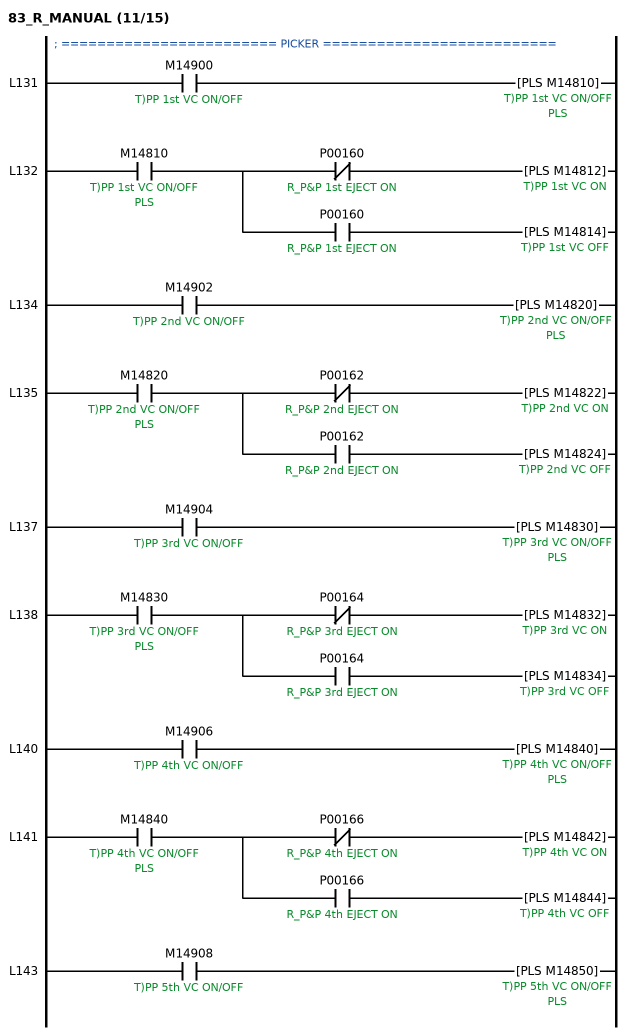
[picture p336: 83_R_MANUAL rungs L131-L143]
// ======================== PICKER ==========================
; L131
LOAD      M14900	// T)PP 1st VC ON/OFF
OUTP      M14810	// T)PP 1st VC ON/OFF PLS
; L132
LOAD      M14810	// T)PP 1st VC ON/OFF PLS
MPUSH
AND NOT   P00160	// R_P&P 1st EJECT ON
OUTP      M14812	// T)PP 1st VC ON
MPOP
AND       P00160	// R_P&P 1st EJECT ON
OUTP      M14814	// T)PP 1st VC OFF
; L134
LOAD      M14902	// T)PP 2nd VC ON/OFF
OUTP      M14820	// T)PP 2nd VC ON/OFF PLS
; L135
LOAD      M14820	// T)PP 2nd VC ON/OFF PLS
MPUSH
AND NOT   P00162	// R_P&P 2nd EJECT ON
OUTP      M14822	// T)PP 2nd VC ON
MPOP
AND       P00162	// R_P&P 2nd EJECT ON
OUTP      M14824	// T)PP 2nd VC OFF
; L137
LOAD      M14904	// T)PP 3rd VC ON/OFF
OUTP      M14830	// T)PP 3rd VC ON/OFF PLS
; L138
LOAD      M14830	// T)PP 3rd VC ON/OFF PLS
MPUSH
AND NOT   P00164	// R_P&P 3rd EJECT ON
OUTP      M14832	// T)PP 3rd VC ON
MPOP
AND       P00164	// R_P&P 3rd EJECT ON
OUTP      M14834	// T)PP 3rd VC OFF
; L140
LOAD      M14906	// T)PP 4th VC ON/OFF
OUTP      M14840	// T)PP 4th VC ON/OFF PLS
; L141
LOAD      M14840	// T)PP 4th VC ON/OFF PLS
MPUSH
AND NOT   P00166	// R_P&P 4th EJECT ON
OUTP      M14842	// T)PP 4th VC ON
MPOP
AND       P00166	// R_P&P 4th EJECT ON
OUTP      M14844	// T)PP 4th VC OFF
; L143
LOAD      M14908	// T)PP 5th VC ON/OFF
OUTP      M14850	// T)PP 5th VC ON/OFF PLS

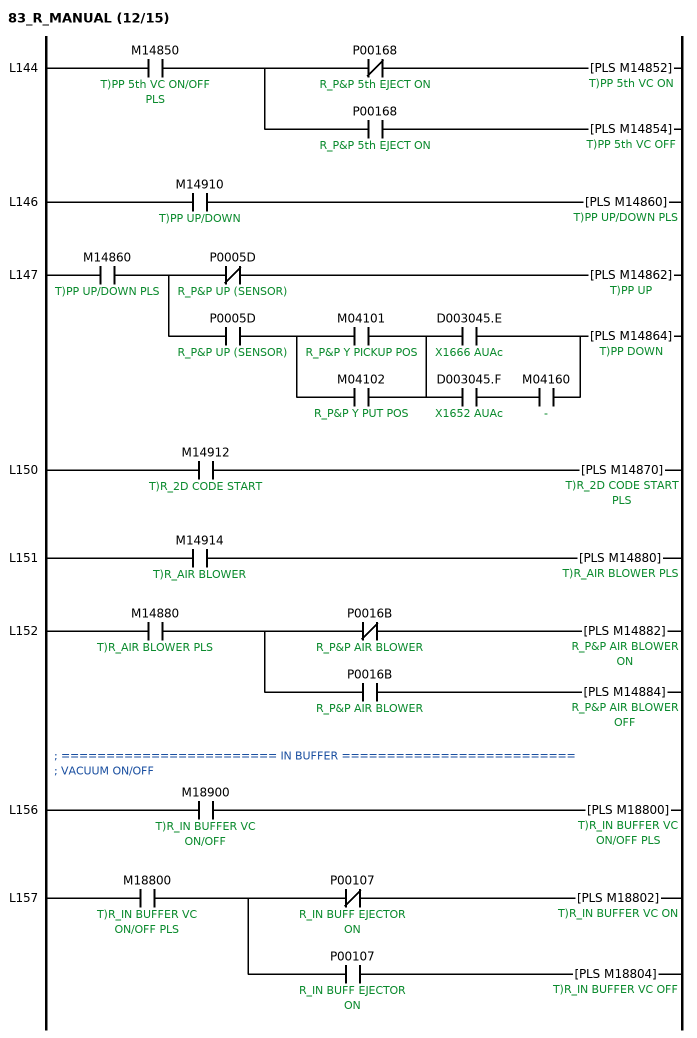
; L144
LOAD      M14850	// T)PP 5th VC ON/OFF PLS
MPUSH
AND NOT   P00168	// R_P&P 5th EJECT ON
OUTP      M14852	// T)PP 5th VC ON
MPOP
AND       P00168	// R_P&P 5th EJECT ON
OUTP      M14854	// T)PP 5th VC OFF
; L146
LOAD      M14910	// T)PP UP/DOWN
OUTP      M14860	// T)PP UP/DOWN PLS
; L147
LOAD      M14860	// T)PP UP/DOWN PLS
MPUSH
AND NOT   P0005D	// R_P&P UP (SENSOR)
OUTP      M14862	// T)PP UP
MPOP
AND       P0005D	// R_P&P UP (SENSOR)
LOAD      M04101	// R_P&P Y PICKUP POS
OR        M04102	// R_P&P Y PUT POS
AND LOAD
LOAD      D003045.E	// X1666 AUAc
LOAD      D003045.F	// X1652 AUAc
AND       M04160	// -
OR LOAD
AND LOAD
OUTP      M14864	// T)PP DOWN
; L150
LOAD      M14912	// T)R_2D CODE START
OUTP      M14870	// T)R_2D CODE START PLS
; L151
LOAD      M14914	// T)R_AIR BLOWER
OUTP      M14880	// T)R_AIR BLOWER PLS
; L152
LOAD      M14880	// T)R_AIR BLOWER PLS
MPUSH
AND NOT   P0016B	// R_P&P AIR BLOWER
OUTP      M14882	// R_P&P AIR BLOWER ON
MPOP
AND       P0016B	// R_P&P AIR BLOWER
OUTP      M14884	// R_P&P AIR BLOWER OFF
// ======================== IN BUFFER ==========================
// VACUUM ON/OFF
; L156
LOAD      M18900	// T)R_IN BUFFER VC ON/OFF
OUTP      M18800	// T)R_IN BUFFER VC ON/OFF PLS
; L157
LOAD      M18800	// T)R_IN BUFFER VC ON/OFF PLS
MPUSH
AND NOT   P00107	// R_IN BUFF EJECTOR ON
OUTP      M18802	// T)R_IN BUFFER VC ON
MPOP
AND       P00107	// R_IN BUFF EJECTOR ON
OUTP      M18804	// T)R_IN BUFFER VC OFF

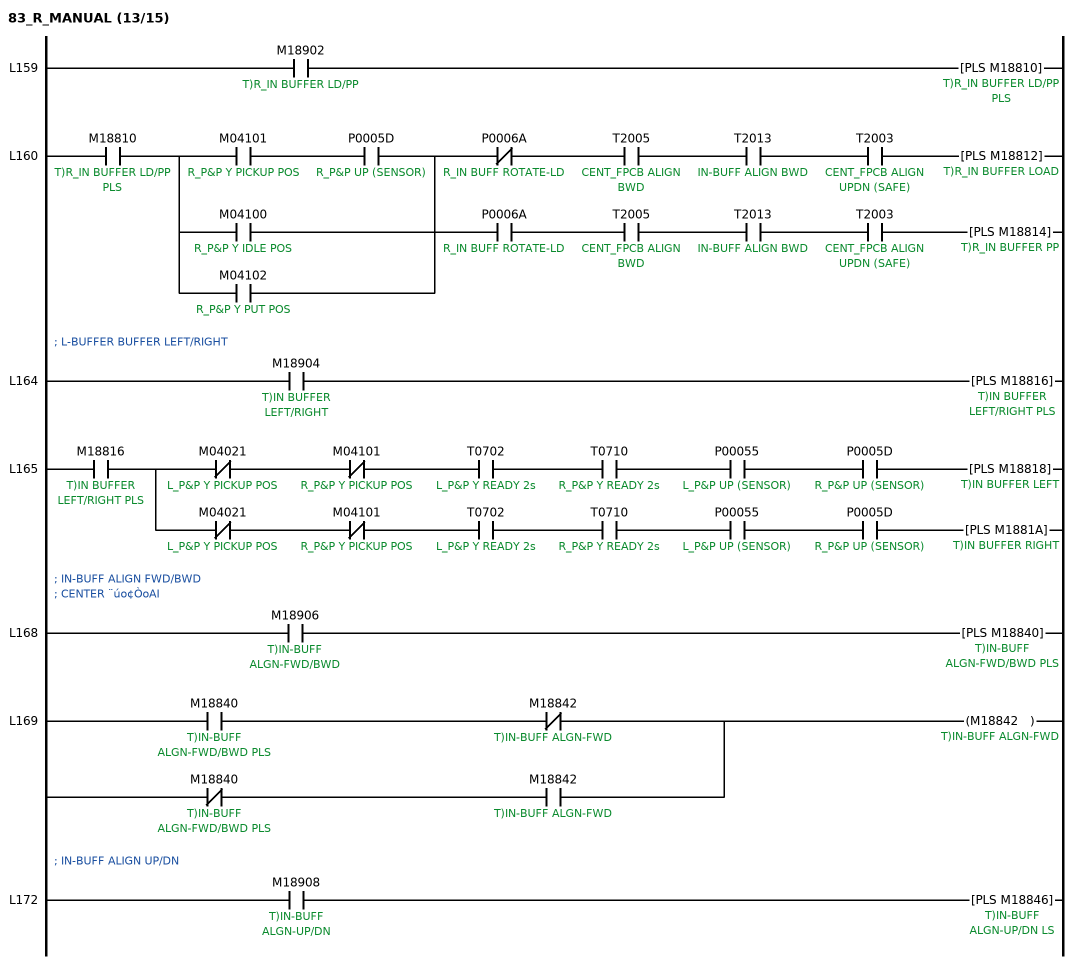
; L159
LOAD      M18902	// T)R_IN BUFFER LD/PP
OUTP      M18810	// T)R_IN BUFFER LD/PP PLS
; L160
LOAD      M18810	// T)R_IN BUFFER LD/PP PLS
LOAD      M04101	// R_P&P Y PICKUP POS
AND       P0005D	// R_P&P UP (SENSOR)
OR        M04100	// R_P&P Y IDLE POS
OR        M04102	// R_P&P Y PUT POS
AND LOAD
MPUSH
AND NOT   P0006A	// R_IN BUFF ROTATE-LD
AND       T2005	// CENT_FPCB ALIGN BWD
AND       T2013	// IN-BUFF ALIGN BWD
AND       T2003	// CENT_FPCB ALIGN UPDN (SAFE)
OUTP      M18812	// T)R_IN BUFFER LOAD
MPOP
AND       P0006A	// R_IN BUFF ROTATE-LD
AND       T2005	// CENT_FPCB ALIGN BWD
AND       T2013	// IN-BUFF ALIGN BWD
AND       T2003	// CENT_FPCB ALIGN UPDN (SAFE)
OUTP      M18814	// T)R_IN BUFFER PP
// L-BUFFER BUFFER LEFT/RIGHT
; L164
LOAD      M18904	// T)IN BUFFER LEFT/RIGHT
OUTP      M18816	// T)IN BUFFER LEFT/RIGHT PLS
; L165
LOAD      M18816	// T)IN BUFFER LEFT/RIGHT PLS
MPUSH
AND NOT   M04021	// L_P&P Y PICKUP POS
AND NOT   M04101	// R_P&P Y PICKUP POS
AND       T0702	// L_P&P Y READY 2s
AND       T0710	// R_P&P Y READY 2s
AND       P00055	// L_P&P UP (SENSOR)
AND       P0005D	// R_P&P UP (SENSOR)
OUTP      M18818	// T)IN BUFFER LEFT
MPOP
AND NOT   M04021	// L_P&P Y PICKUP POS
AND NOT   M04101	// R_P&P Y PICKUP POS
AND       T0702	// L_P&P Y READY 2s
AND       T0710	// R_P&P Y READY 2s
AND       P00055	// L_P&P UP (SENSOR)
AND       P0005D	// R_P&P UP (SENSOR)
OUTP      M1881A	// T)IN BUFFER RIGHT
// IN-BUFF ALIGN FWD/BWD
; L168
LOAD      M18906	// T)IN-BUFF ALGN-FWD/BWD
OUTP      M18840	// T)IN-BUFF ALGN-FWD/BWD PLS
// output comment: CENTER ¨úo¢ÒoAI
; L169
LOAD      M18840	// T)IN-BUFF ALGN-FWD/BWD PLS
AND NOT   M18842	// T)IN-BUFF ALGN-FWD
LOAD NOT  M18840	// T)IN-BUFF ALGN-FWD/BWD PLS
AND       M18842	// T)IN-BUFF ALGN-FWD
OR LOAD
OUT       M18842	// T)IN-BUFF ALGN-FWD
// IN-BUFF ALIGN UP/DN
; L172
LOAD      M18908	// T)IN-BUFF ALGN-UP/DN
OUTP      M18846	// T)IN-BUFF ALGN-UP/DN LS

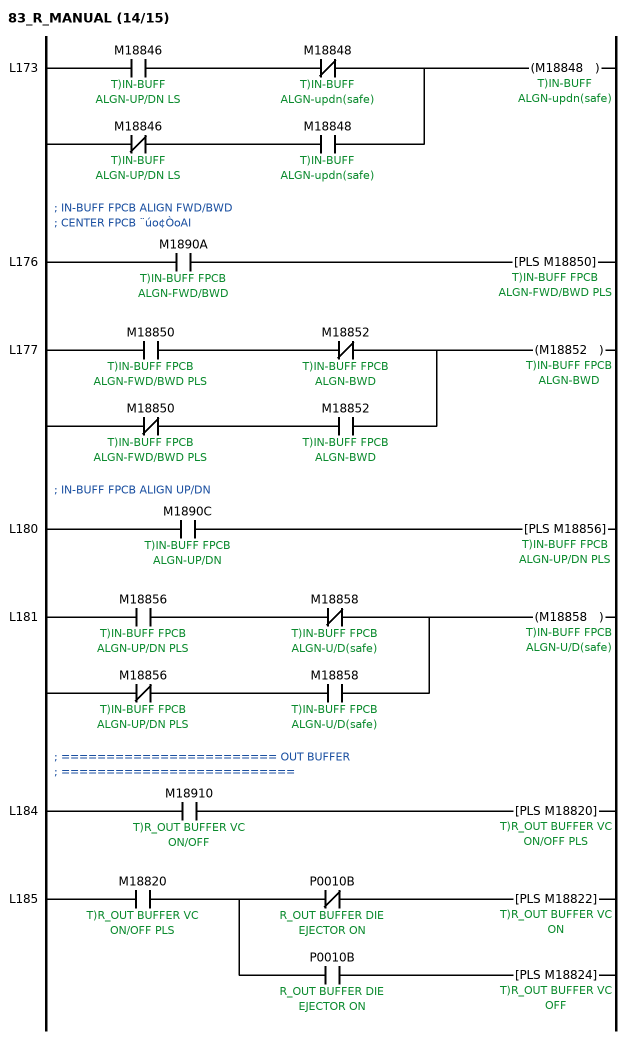
; L173
LOAD      M18846	// T)IN-BUFF ALGN-UP/DN LS
AND NOT   M18848	// T)IN-BUFF ALGN-updn(safe)
LOAD NOT  M18846	// T)IN-BUFF ALGN-UP/DN LS
AND       M18848	// T)IN-BUFF ALGN-updn(safe)
OR LOAD
OUT       M18848	// T)IN-BUFF ALGN-updn(safe)
// IN-BUFF FPCB ALIGN FWD/BWD
; L176
LOAD      M1890A	// T)IN-BUFF FPCB ALGN-FWD/BWD
OUTP      M18850	// T)IN-BUFF FPCB ALGN-FWD/BWD PLS
// output comment: CENTER FPCB ¨úo¢ÒoAI
; L177
LOAD      M18850	// T)IN-BUFF FPCB ALGN-FWD/BWD PLS
AND NOT   M18852	// T)IN-BUFF FPCB ALGN-BWD
LOAD NOT  M18850	// T)IN-BUFF FPCB ALGN-FWD/BWD PLS
AND       M18852	// T)IN-BUFF FPCB ALGN-BWD
OR LOAD
OUT       M18852	// T)IN-BUFF FPCB ALGN-BWD
// IN-BUFF FPCB ALIGN UP/DN
; L180
LOAD      M1890C	// T)IN-BUFF FPCB ALGN-UP/DN
OUTP      M18856	// T)IN-BUFF FPCB ALGN-UP/DN PLS
; L181
LOAD      M18856	// T)IN-BUFF FPCB ALGN-UP/DN PLS
AND NOT   M18858	// T)IN-BUFF FPCB ALGN-U/D(safe)
LOAD NOT  M18856	// T)IN-BUFF FPCB ALGN-UP/DN PLS
AND       M18858	// T)IN-BUFF FPCB ALGN-U/D(safe)
OR LOAD
OUT       M18858	// T)IN-BUFF FPCB ALGN-U/D(safe)
// ======================== OUT BUFFER ==========================
; L184
LOAD      M18910	// T)R_OUT BUFFER VC ON/OFF
OUTP      M18820	// T)R_OUT BUFFER VC ON/OFF PLS
; L185
LOAD      M18820	// T)R_OUT BUFFER VC ON/OFF PLS
MPUSH
AND NOT   P0010B	// R_OUT BUFFER DIE EJECTOR ON
OUTP      M18822	// T)R_OUT BUFFER VC ON
MPOP
AND       P0010B	// R_OUT BUFFER DIE EJECTOR ON
OUTP      M18824	// T)R_OUT BUFFER VC OFF

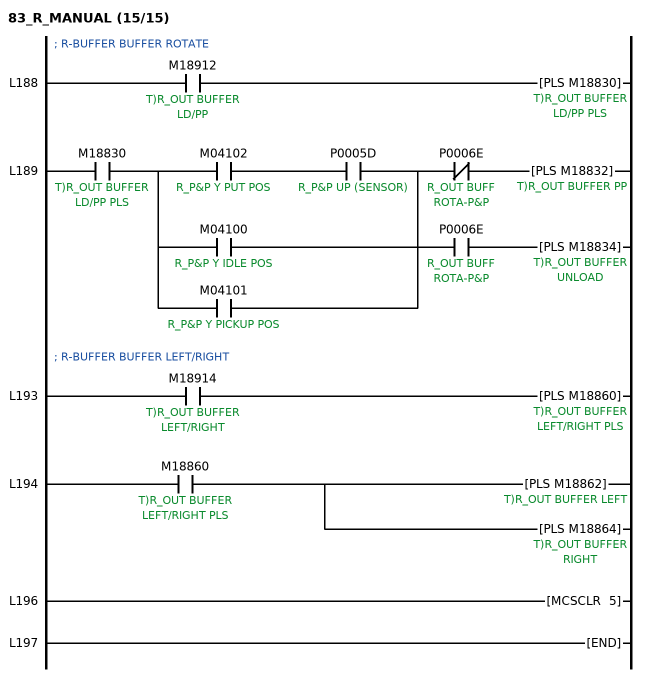
// R-BUFFER BUFFER ROTATE
; L188
LOAD      M18912	// T)R_OUT BUFFER LD/PP
OUTP      M18830	// T)R_OUT BUFFER LD/PP PLS
; L189
LOAD      M18830	// T)R_OUT BUFFER LD/PP PLS
LOAD      M04102	// R_P&P Y PUT POS
AND       P0005D	// R_P&P UP (SENSOR)
OR        M04100	// R_P&P Y IDLE POS
OR        M04101	// R_P&P Y PICKUP POS
AND LOAD
MPUSH
AND NOT   P0006E	// R_OUT BUFF ROTA-P&P
OUTP      M18832	// T)R_OUT BUFFER PP
MPOP
AND       P0006E	// R_OUT BUFF ROTA-P&P
OUTP      M18834	// T)R_OUT BUFFER UNLOAD
// R-BUFFER BUFFER LEFT/RIGHT
; L193
LOAD      M18914	// T)R_OUT BUFFER LEFT/RIGHT
OUTP      M18860	// T)R_OUT BUFFER LEFT/RIGHT PLS
; L194
LOAD      M18860	// T)R_OUT BUFFER LEFT/RIGHT PLS
OUTP      M18862	// T)R_OUT BUFFER LEFT
OUTP      M18864	// T)R_OUT BUFFER RIGHT
; L196
MCSCLR    5
; L197
END

PROGRAM 84_RUN_TIME (task: ¨ö¨¬A¥ì CA¡¤I¡¾¡¿¡¤¡Í)

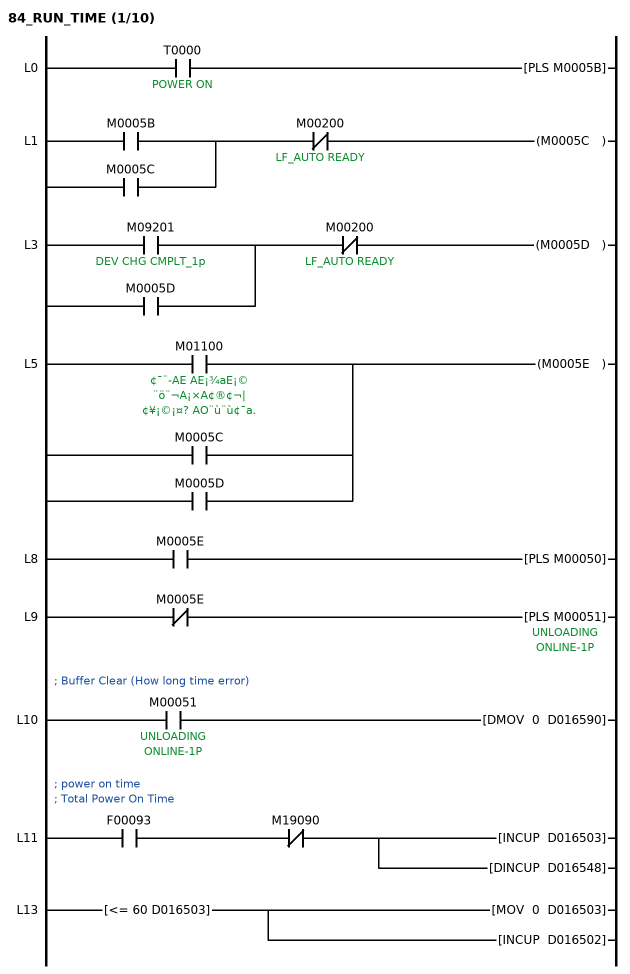
; L0
LOAD      T0000	// POWER ON
OUTP      M0005B
; L1
LOAD      M0005B
OR        M0005C
AND NOT   M00200	// LF_AUTO READY
OUT       M0005C
; L3
LOAD      M09201	// DEV CHG CMPLT_1p
OR        M0005D
AND NOT   M00200	// LF_AUTO READY
OUT       M0005D
; L5
LOAD      M01100	// ¢¯¨­AE AE¡¾aE¡© ¨ö¨¬A¡×A¢®¢¬| ¢¥¡©¡¤? AO¨ù¨ù¢¯a.
OR        M0005C
OR        M0005D
OUT       M0005E
; L8
LOAD      M0005E
OUTP      M00050
; L9
LOAD NOT  M0005E
OUTP      M00051	// UNLOADING ONLINE-1P
; L10
LOAD      M00051	// UNLOADING ONLINE-1P
DMOV      0 D016590
// output comment: Buffer Clear (How long time error)
; L11
LOAD      F00093
AND NOT   M19090
INCUP     D016503
DINCUP    D016548
// output comment: power on time
// output comment: Total Power On Time
; L13
LOAD<=    60 D016503
MOV       0 D016503
INCUP     D016502

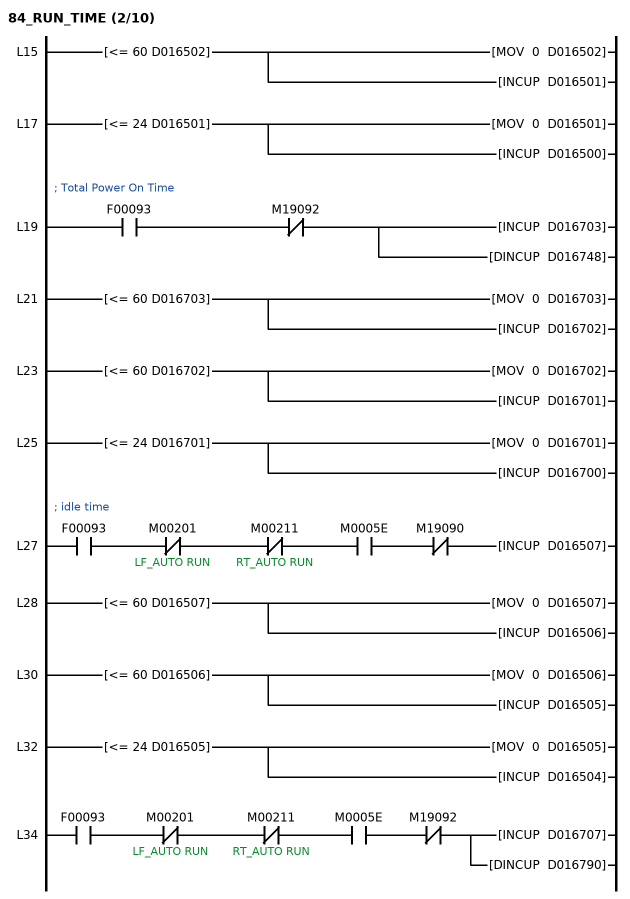
; L15
LOAD<=    60 D016502
MOV       0 D016502
INCUP     D016501
; L17
LOAD<=    24 D016501
MOV       0 D016501
INCUP     D016500
; L19
LOAD      F00093
AND NOT   M19092
INCUP     D016703
DINCUP    D016748
// output comment: Total Power On Time
; L21
LOAD<=    60 D016703
MOV       0 D016703
INCUP     D016702
; L23
LOAD<=    60 D016702
MOV       0 D016702
INCUP     D016701
; L25
LOAD<=    24 D016701
MOV       0 D016701
INCUP     D016700
; L27
LOAD      F00093
AND NOT   M00201	// LF_AUTO RUN
AND NOT   M00211	// RT_AUTO RUN
AND       M0005E
AND NOT   M19090
INCUP     D016507
// output comment: idle time
; L28
LOAD<=    60 D016507
MOV       0 D016507
INCUP     D016506
; L30
LOAD<=    60 D016506
MOV       0 D016506
INCUP     D016505
; L32
LOAD<=    24 D016505
MOV       0 D016505
INCUP     D016504
; L34
LOAD      F00093
AND NOT   M00201	// LF_AUTO RUN
AND NOT   M00211	// RT_AUTO RUN
AND       M0005E
AND NOT   M19092
INCUP     D016707
DINCUP    D016790

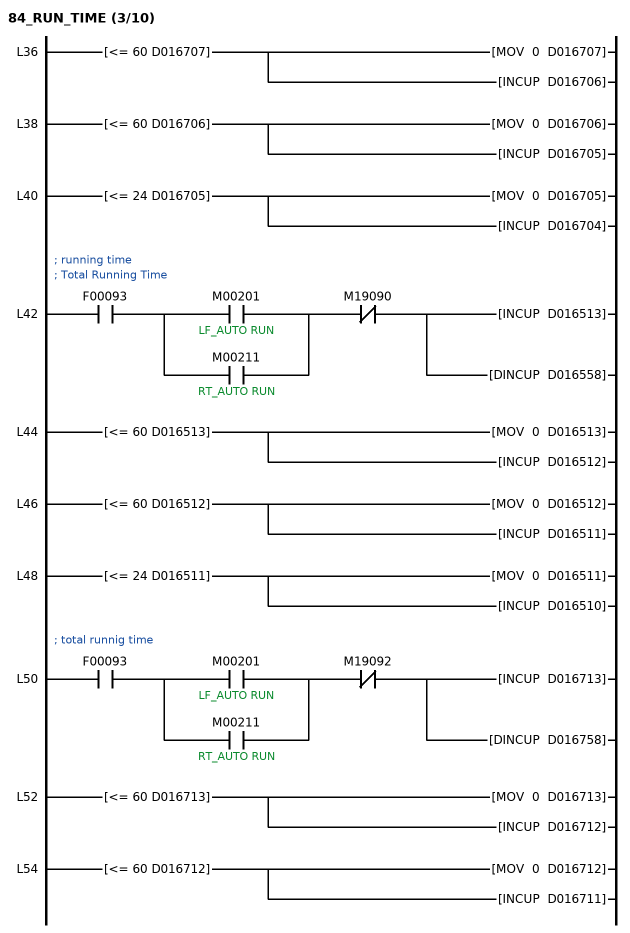
; L36
LOAD<=    60 D016707
MOV       0 D016707
INCUP     D016706
; L38
LOAD<=    60 D016706
MOV       0 D016706
INCUP     D016705
; L40
LOAD<=    24 D016705
MOV       0 D016705
INCUP     D016704
; L42
LOAD      F00093
LOAD      M00201	// LF_AUTO RUN
OR        M00211	// RT_AUTO RUN
AND LOAD
AND NOT   M19090
INCUP     D016513
DINCUP    D016558
// output comment: running time
// output comment: Total Running Time
; L44
LOAD<=    60 D016513
MOV       0 D016513
INCUP     D016512
; L46
LOAD<=    60 D016512
MOV       0 D016512
INCUP     D016511
; L48
LOAD<=    24 D016511
MOV       0 D016511
INCUP     D016510
; L50
LOAD      F00093
LOAD      M00201	// LF_AUTO RUN
OR        M00211	// RT_AUTO RUN
AND LOAD
AND NOT   M19092
INCUP     D016713
DINCUP    D016758
// output comment: total runnig time
; L52
LOAD<=    60 D016713
MOV       0 D016713
INCUP     D016712
; L54
LOAD<=    60 D016712
MOV       0 D016712
INCUP     D016711

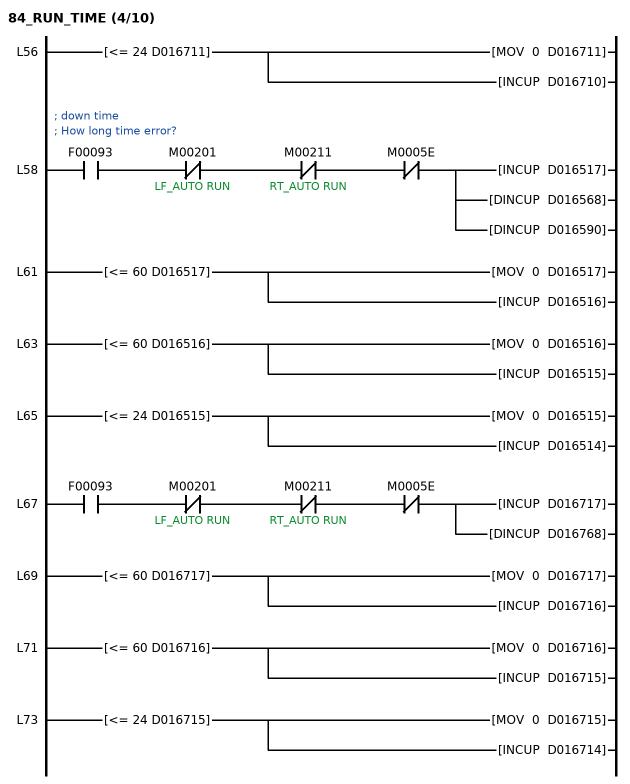
; L56
LOAD<=    24 D016711
MOV       0 D016711
INCUP     D016710
; L58
LOAD      F00093
AND NOT   M00201	// LF_AUTO RUN
AND NOT   M00211	// RT_AUTO RUN
AND NOT   M0005E
INCUP     D016517
DINCUP    D016568
DINCUP    D016590
// output comment: down time
// output comment: How long time error?
; L61
LOAD<=    60 D016517
MOV       0 D016517
INCUP     D016516
; L63
LOAD<=    60 D016516
MOV       0 D016516
INCUP     D016515
; L65
LOAD<=    24 D016515
MOV       0 D016515
INCUP     D016514
; L67
LOAD      F00093
AND NOT   M00201	// LF_AUTO RUN
AND NOT   M00211	// RT_AUTO RUN
AND NOT   M0005E
INCUP     D016717
DINCUP    D016768
; L69
LOAD<=    60 D016717
MOV       0 D016717
INCUP     D016716
; L71
LOAD<=    60 D016716
MOV       0 D016716
INCUP     D016715
; L73
LOAD<=    24 D016715
MOV       0 D016715
INCUP     D016714

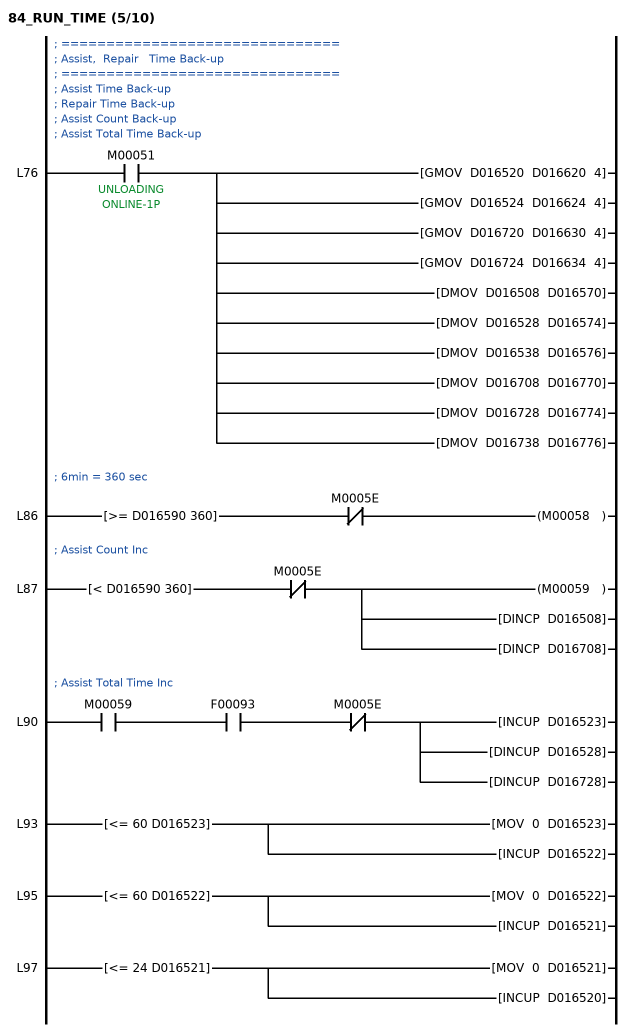
// ===============================
// Assist,  Repair   Time Back-up
// ===============================
; L76
LOAD      M00051	// UNLOADING ONLINE-1P
GMOV      D016520 D016620 4
GMOV      D016524 D016624 4
GMOV      D016720 D016630 4
GMOV      D016724 D016634 4
DMOV      D016508 D016570
DMOV      D016528 D016574
DMOV      D016538 D016576
DMOV      D016708 D016770
DMOV      D016728 D016774
DMOV      D016738 D016776
// output comment: Assist Time Back-up
// output comment: Repair Time Back-up
// output comment: Assist Count Back-up
// output comment: Assist Total Time Back-up
; L86
LOAD>=    D016590 360
AND NOT   M0005E
OUT       M00058
// output comment: 6min = 360 sec
; L87
LOAD<     D016590 360
AND NOT   M0005E
OUT       M00059
DINCP     D016508
DINCP     D016708
// output comment: Assist Count Inc
; L90
LOAD      M00059
AND       F00093
AND NOT   M0005E
INCUP     D016523
DINCUP    D016528
DINCUP    D016728
// output comment: Assist Total Time Inc
; L93
LOAD<=    60 D016523
MOV       0 D016523
INCUP     D016522
; L95
LOAD<=    60 D016522
MOV       0 D016522
INCUP     D016521
; L97
LOAD<=    24 D016521
MOV       0 D016521
INCUP     D016520

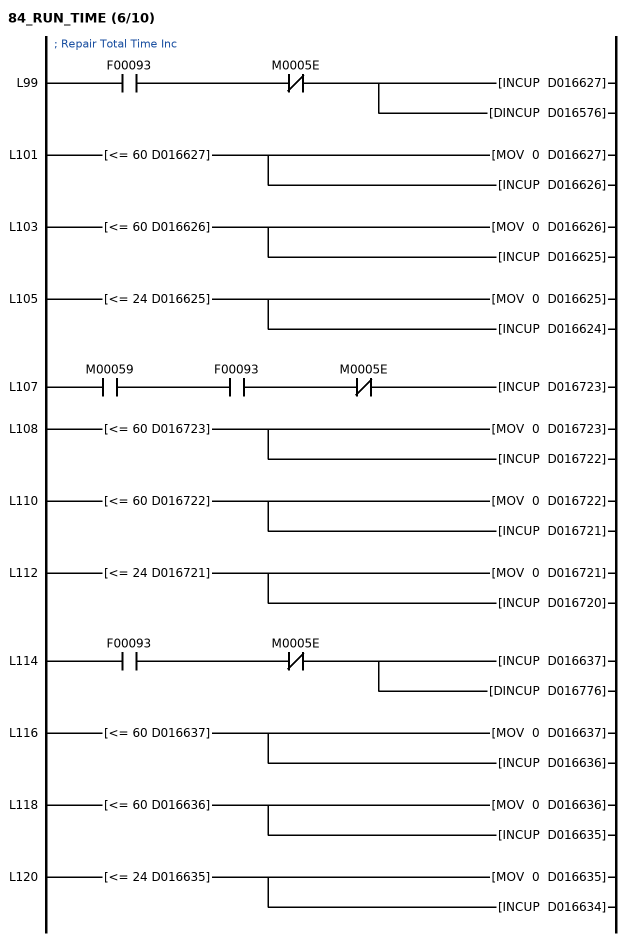
; L99
LOAD      F00093
AND NOT   M0005E
INCUP     D016627
DINCUP    D016576
// output comment: Repair Total Time Inc
; L101
LOAD<=    60 D016627
MOV       0 D016627
INCUP     D016626
; L103
LOAD<=    60 D016626
MOV       0 D016626
INCUP     D016625
; L105
LOAD<=    24 D016625
MOV       0 D016625
INCUP     D016624
; L107
LOAD      M00059
AND       F00093
AND NOT   M0005E
INCUP     D016723
; L108
LOAD<=    60 D016723
MOV       0 D016723
INCUP     D016722
; L110
LOAD<=    60 D016722
MOV       0 D016722
INCUP     D016721
; L112
LOAD<=    24 D016721
MOV       0 D016721
INCUP     D016720
; L114
LOAD      F00093
AND NOT   M0005E
INCUP     D016637
DINCUP    D016776
; L116
LOAD<=    60 D016637
MOV       0 D016637
INCUP     D016636
; L118
LOAD<=    60 D016636
MOV       0 D016636
INCUP     D016635
; L120
LOAD<=    24 D016635
MOV       0 D016635
INCUP     D016634

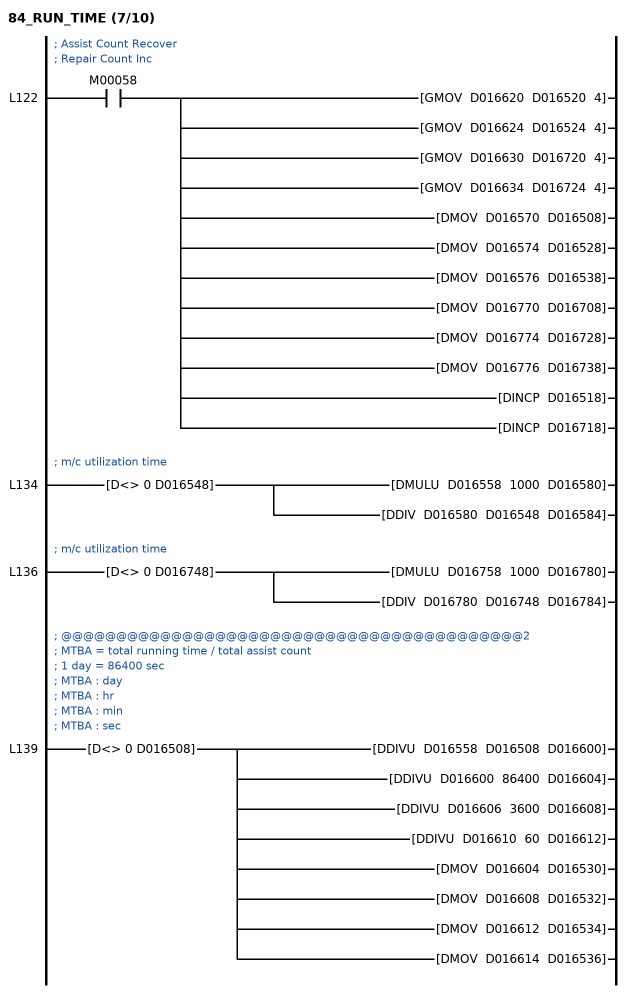
; L122
LOAD      M00058
GMOV      D016620 D016520 4
GMOV      D016624 D016524 4
GMOV      D016630 D016720 4
GMOV      D016634 D016724 4
DMOV      D016570 D016508
DMOV      D016574 D016528
DMOV      D016576 D016538
DMOV      D016770 D016708
DMOV      D016774 D016728
DMOV      D016776 D016738
DINCP     D016518
DINCP     D016718
// output comment: Assist Count Recover
// output comment: Repair Count Inc
; L134
LOADD<>   0 D016548
DMULU     D016558 1000 D016580
DDIV      D016580 D016548 D016584
// output comment: m/c utilization time
; L136
LOADD<>   0 D016748
DMULU     D016758 1000 D016780
DDIV      D016780 D016748 D016784
// output comment: m/c utilization time
// @@@@@@@@@@@@@@@@@@@@@@@@@@@@@@@@@@@@@@@@@@2
; L139
LOADD<>   0 D016508
DDIVU     D016558 D016508 D016600
DDIVU     D016600 86400 D016604
DDIVU     D016606 3600 D016608
DDIVU     D016610 60 D016612
DMOV      D016604 D016530
DMOV      D016608 D016532
DMOV      D016612 D016534
DMOV      D016614 D016536
// output comment: MTBA = total running time / total assist count
// output comment: 1 day = 86400 sec
// output comment: MTBA : day
// output comment: MTBA : hr
// output comment: MTBA : min
// output comment: MTBA : sec

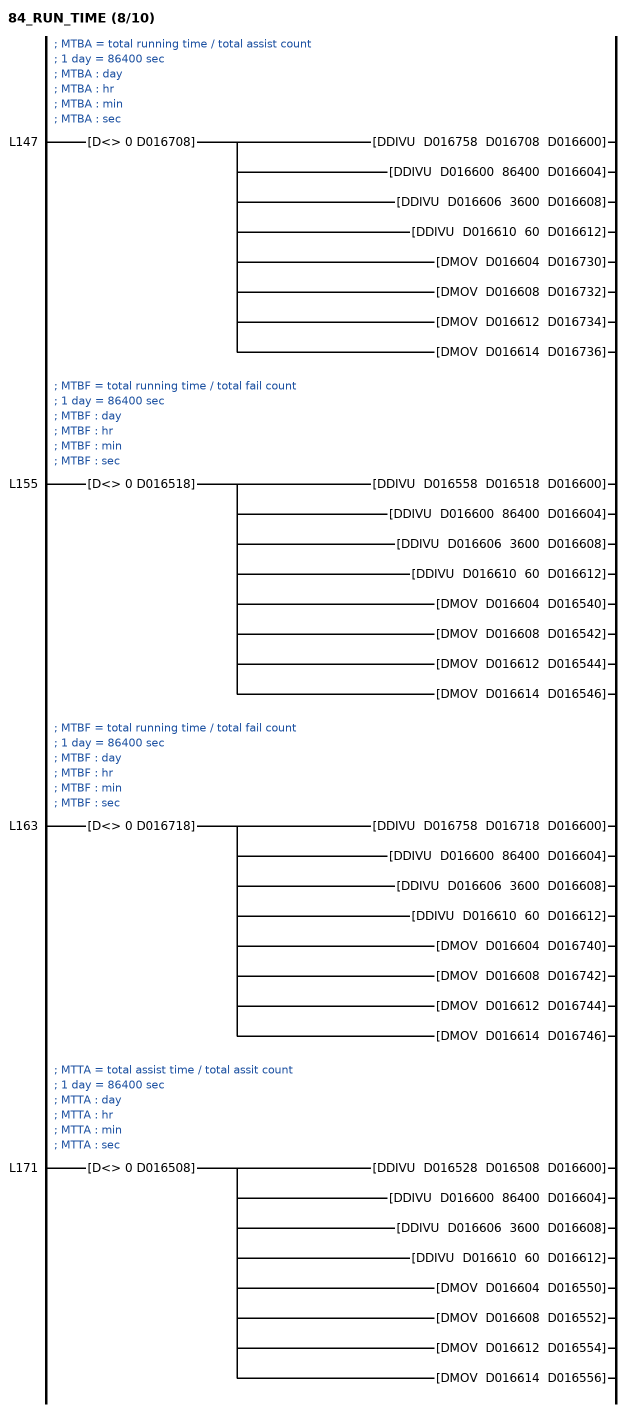
; L147
LOADD<>   0 D016708
DDIVU     D016758 D016708 D016600
DDIVU     D016600 86400 D016604
DDIVU     D016606 3600 D016608
DDIVU     D016610 60 D016612
DMOV      D016604 D016730
DMOV      D016608 D016732
DMOV      D016612 D016734
DMOV      D016614 D016736
// output comment: MTBA = total running time / total assist count
// output comment: 1 day = 86400 sec
// output comment: MTBA : day
// output comment: MTBA : hr
// output comment: MTBA : min
// output comment: MTBA : sec
; L155
LOADD<>   0 D016518
DDIVU     D016558 D016518 D016600
DDIVU     D016600 86400 D016604
DDIVU     D016606 3600 D016608
DDIVU     D016610 60 D016612
DMOV      D016604 D016540
DMOV      D016608 D016542
DMOV      D016612 D016544
DMOV      D016614 D016546
// output comment: MTBF = total running time / total fail count
// output comment: 1 day = 86400 sec
// output comment: MTBF : day
// output comment: MTBF : hr
// output comment: MTBF : min
// output comment: MTBF : sec
; L163
LOADD<>   0 D016718
DDIVU     D016758 D016718 D016600
DDIVU     D016600 86400 D016604
DDIVU     D016606 3600 D016608
DDIVU     D016610 60 D016612
DMOV      D016604 D016740
DMOV      D016608 D016742
DMOV      D016612 D016744
DMOV      D016614 D016746
// output comment: MTBF = total running time / total fail count
// output comment: 1 day = 86400 sec
// output comment: MTBF : day
// output comment: MTBF : hr
// output comment: MTBF : min
// output comment: MTBF : sec
; L171
LOADD<>   0 D016508
DDIVU     D016528 D016508 D016600
DDIVU     D016600 86400 D016604
DDIVU     D016606 3600 D016608
DDIVU     D016610 60 D016612
DMOV      D016604 D016550
DMOV      D016608 D016552
DMOV      D016612 D016554
DMOV      D016614 D016556
// output comment: MTTA = total assist time / total assit count
// output comment: 1 day = 86400 sec
// output comment: MTTA : day
// output comment: MTTA : hr
// output comment: MTTA : min
// output comment: MTTA : sec

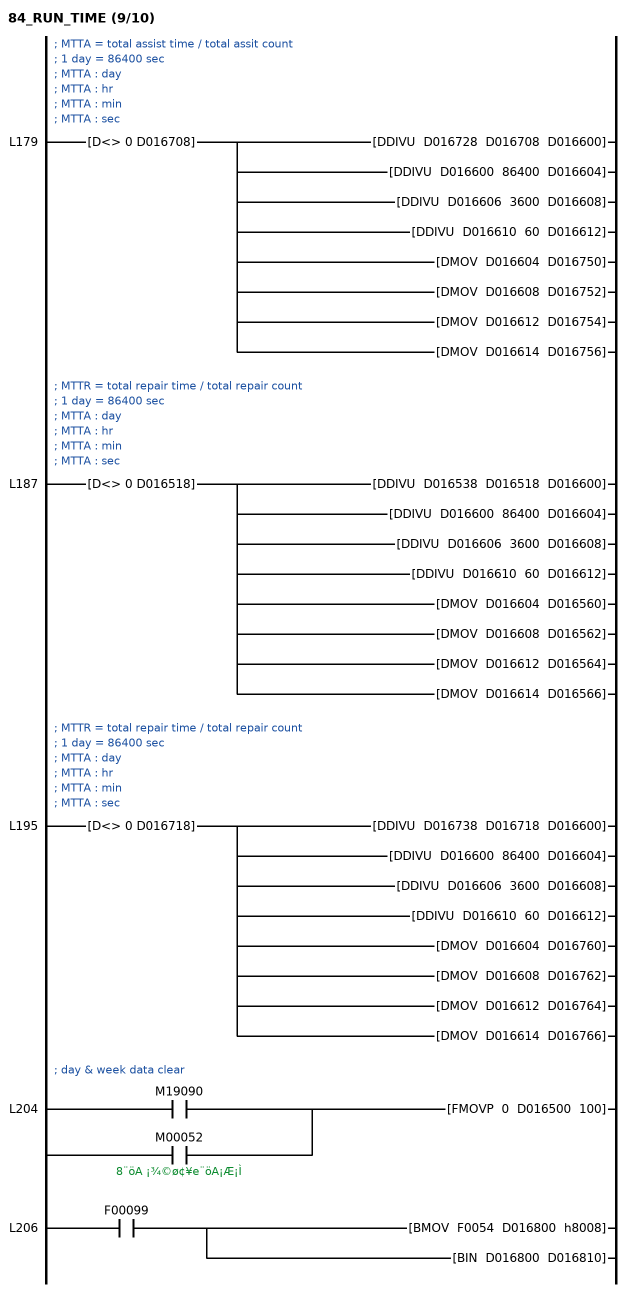
; L179
LOADD<>   0 D016708
DDIVU     D016728 D016708 D016600
DDIVU     D016600 86400 D016604
DDIVU     D016606 3600 D016608
DDIVU     D016610 60 D016612
DMOV      D016604 D016750
DMOV      D016608 D016752
DMOV      D016612 D016754
DMOV      D016614 D016756
// output comment: MTTA = total assist time / total assit count
// output comment: 1 day = 86400 sec
// output comment: MTTA : day
// output comment: MTTA : hr
// output comment: MTTA : min
// output comment: MTTA : sec
; L187
LOADD<>   0 D016518
DDIVU     D016538 D016518 D016600
DDIVU     D016600 86400 D016604
DDIVU     D016606 3600 D016608
DDIVU     D016610 60 D016612
DMOV      D016604 D016560
DMOV      D016608 D016562
DMOV      D016612 D016564
DMOV      D016614 D016566
// output comment: MTTR = total repair time / total repair count
// output comment: 1 day = 86400 sec
// output comment: MTTA : day
// output comment: MTTA : hr
// output comment: MTTA : min
// output comment: MTTA : sec
; L195
LOADD<>   0 D016718
DDIVU     D016738 D016718 D016600
DDIVU     D016600 86400 D016604
DDIVU     D016606 3600 D016608
DDIVU     D016610 60 D016612
DMOV      D016604 D016760
DMOV      D016608 D016762
DMOV      D016612 D016764
DMOV      D016614 D016766
// output comment: MTTR = total repair time / total repair count
// output comment: 1 day = 86400 sec
// output comment: MTTA : day
// output comment: MTTA : hr
// output comment: MTTA : min
// output comment: MTTA : sec
// day & week data clear
; L204
LOAD      M19090
OR        M00052	// 8¨öA ¡¾©ø¢¥e¨öA¡Æ¡Ì
FMOVP     0 D016500 100
; L206
LOAD      F00099
BMOV      F0054 D016800 h8008
BIN       D016800 D016810

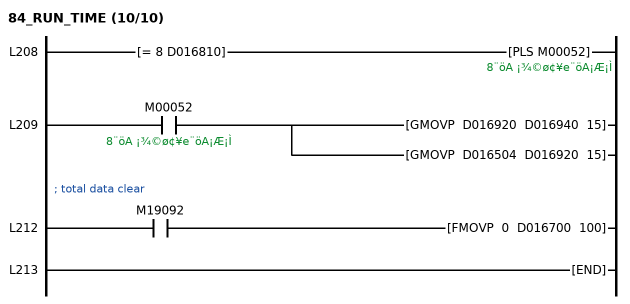
; L208
LOAD=     8 D016810
OUTP      M00052	// 8¨öA ¡¾©ø¢¥e¨öA¡Æ¡Ì
; L209
LOAD      M00052	// 8¨öA ¡¾©ø¢¥e¨öA¡Æ¡Ì
GMOVP     D016920 D016940 15
GMOVP     D016504 D016920 15
// total data clear
; L212
LOAD      M19092
FMOVP     0 D016700 100
; L213
END

PROGRAM 90_ALARM (task: ¨ö¨¬A¥ì CA¡¤I¡¾¡¿¡¤¡Í)

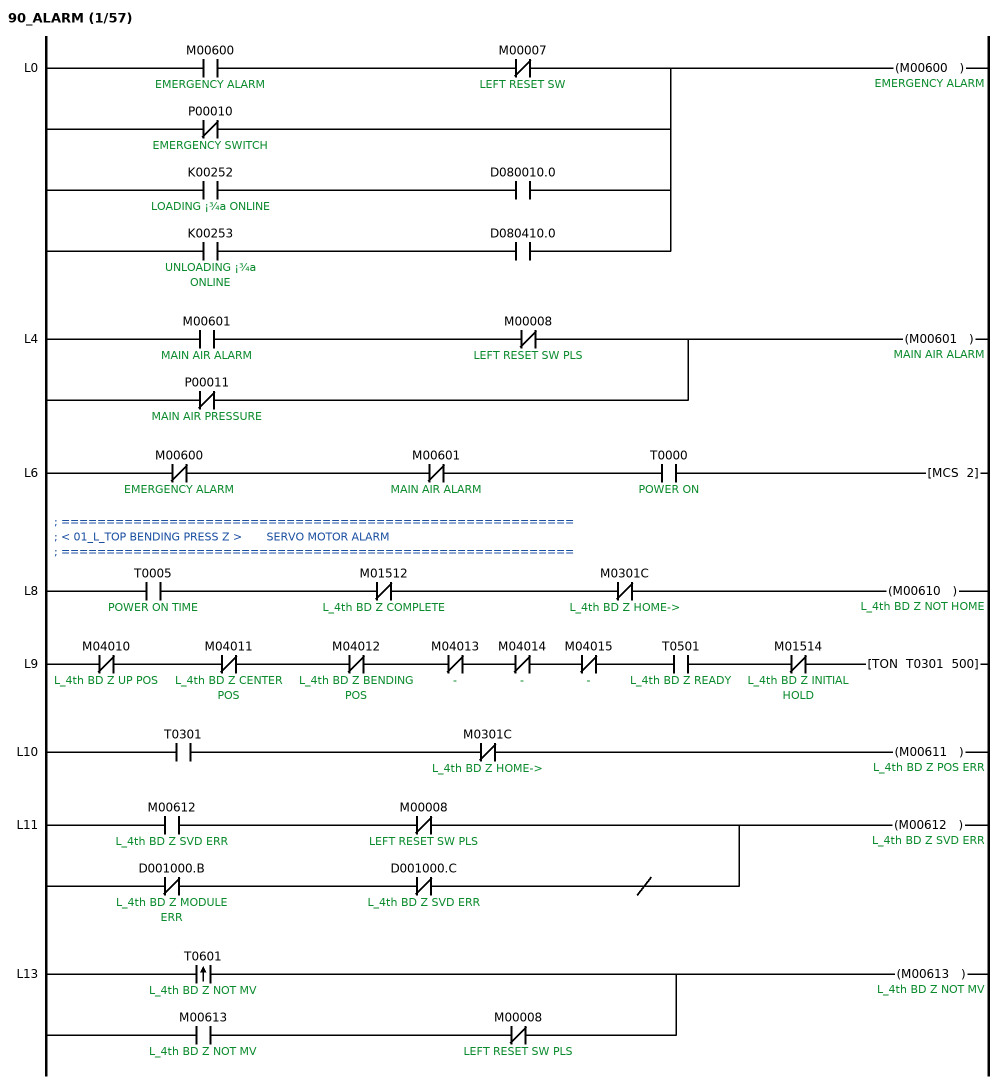
; L0
LOAD      M00600	// EMERGENCY ALARM
AND NOT   M00007	// LEFT RESET SW
OR NOT    P00010	// EMERGENCY SWITCH
LOAD      K00252	// LOADING ¡¾a ONLINE
AND       D080010.0
OR LOAD
LOAD      K00253	// UNLOADING ¡¾a ONLINE
AND       D080410.0
OR LOAD
OUT       M00600	// EMERGENCY ALARM
; L4
LOAD      M00601	// MAIN AIR ALARM
AND NOT   M00008	// LEFT RESET SW PLS
OR NOT    P00011	// MAIN AIR PRESSURE
OUT       M00601	// MAIN AIR ALARM
; L6
LOAD NOT  M00600	// EMERGENCY ALARM
AND NOT   M00601	// MAIN AIR ALARM
AND       T0000	// POWER ON
MCS       2
// =========================================================
// 
//        < 01_L_TOP BENDING PRESS Z >       SERVO MOTOR ALARM
// 
// =========================================================
; L8
LOAD      T0005	// POWER ON TIME
AND NOT   M01512	// L_4th BD Z COMPLETE
AND NOT   M0301C	// L_4th BD Z HOME->
OUT       M00610	// L_4th BD Z NOT HOME
; L9
LOAD NOT  M04010	// L_4th BD Z UP POS
AND NOT   M04011	// L_4th BD Z CENTER POS
AND NOT   M04012	// L_4th BD Z BENDING POS
AND NOT   M04013	// -
AND NOT   M04014	// -
AND NOT   M04015	// -
AND       T0501	// L_4th BD Z READY
AND NOT   M01514	// L_4th BD Z INITIAL HOLD
TON       T0301 500
; L10
LOAD      T0301
AND NOT   M0301C	// L_4th BD Z HOME->
OUT       M00611	// L_4th BD Z POS ERR
; L11
LOAD      M00612	// L_4th BD Z SVD ERR
AND NOT   M00008	// LEFT RESET SW PLS
LOAD NOT  D001000.B	// L_4th BD Z MODULE ERR
AND NOT   D001000.C	// L_4th BD Z SVD ERR
NOT
OR LOAD
OUT       M00612	// L_4th BD Z SVD ERR
; L13
LOADP     T0601	// L_4th BD Z NOT MV
LOAD      M00613	// L_4th BD Z NOT MV
AND NOT   M00008	// LEFT RESET SW PLS
OR LOAD
OUT       M00613	// L_4th BD Z NOT MV

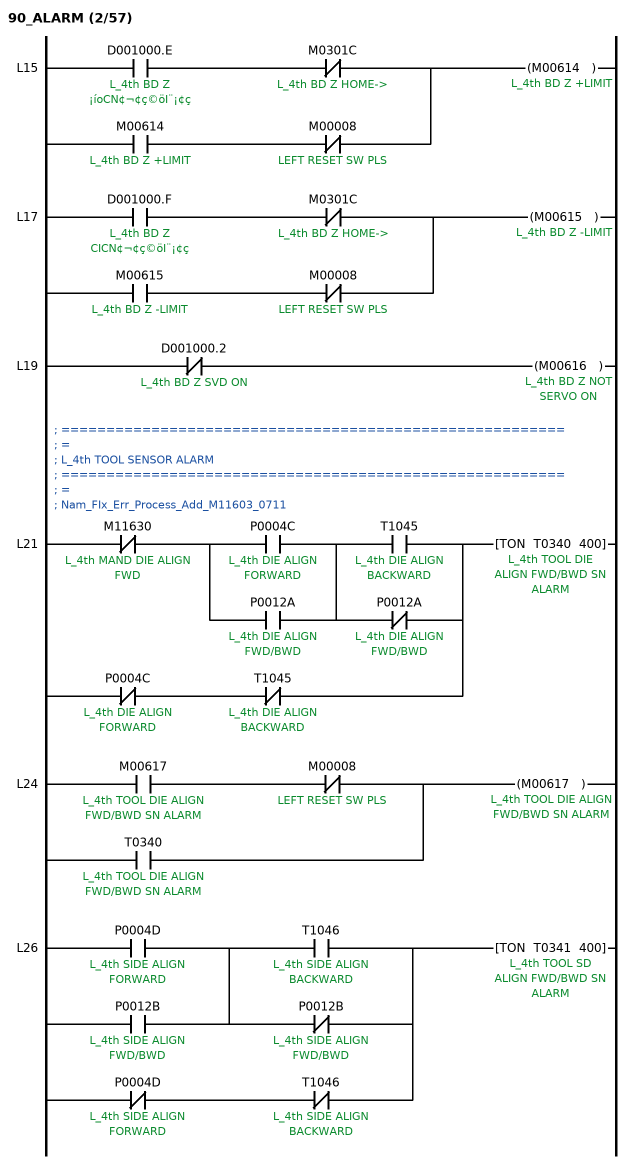
; L15
LOAD      D001000.E	// L_4th BD Z ¡íoCN¢¬¢ç©öI¨¡¢ç
AND NOT   M0301C	// L_4th BD Z HOME->
LOAD      M00614	// L_4th BD Z +LIMIT
AND NOT   M00008	// LEFT RESET SW PLS
OR LOAD
OUT       M00614	// L_4th BD Z +LIMIT
; L17
LOAD      D001000.F	// L_4th BD Z CICN¢¬¢ç©öI¨¡¢ç
AND NOT   M0301C	// L_4th BD Z HOME->
LOAD      M00615	// L_4th BD Z -LIMIT
AND NOT   M00008	// LEFT RESET SW PLS
OR LOAD
OUT       M00615	// L_4th BD Z -LIMIT
; L19
LOAD NOT  D001000.2	// L_4th BD Z SVD ON
OUT       M00616	// L_4th BD Z NOT SERVO ON
// =========================================================
// 
//        L_4th TOOL SENSOR ALARM
// 
// =========================================================
; L21
LOAD NOT  M11630	// L_4th MAND DIE ALIGN FWD
LOAD      P0004C	// L_4th DIE ALIGN FORWARD
OR        P0012A	// L_4th DIE ALIGN FWD/BWD
AND LOAD
LOAD      T1045	// L_4th DIE ALIGN BACKWARD
OR NOT    P0012A	// L_4th DIE ALIGN FWD/BWD
AND LOAD
LOAD NOT  P0004C	// L_4th DIE ALIGN FORWARD
AND NOT   T1045	// L_4th DIE ALIGN BACKWARD
OR LOAD
TON       T0340 400	// L_4th TOOL DIE ALIGN FWD/BWD SN ALARM
// output comment: Nam_FIx_Err_Process_Add_M11603_0711
; L24
LOAD      M00617	// L_4th TOOL DIE ALIGN FWD/BWD SN ALARM
AND NOT   M00008	// LEFT RESET SW PLS
OR        T0340	// L_4th TOOL DIE ALIGN FWD/BWD SN ALARM
OUT       M00617	// L_4th TOOL DIE ALIGN FWD/BWD SN ALARM
; L26
LOAD      P0004D	// L_4th SIDE ALIGN FORWARD
OR        P0012B	// L_4th SIDE ALIGN FWD/BWD
LOAD      T1046	// L_4th SIDE ALIGN BACKWARD
OR NOT    P0012B	// L_4th SIDE ALIGN FWD/BWD
AND LOAD
LOAD NOT  P0004D	// L_4th SIDE ALIGN FORWARD
AND NOT   T1046	// L_4th SIDE ALIGN BACKWARD
OR LOAD
TON       T0341 400	// L_4th TOOL SD ALIGN FWD/BWD SN ALARM

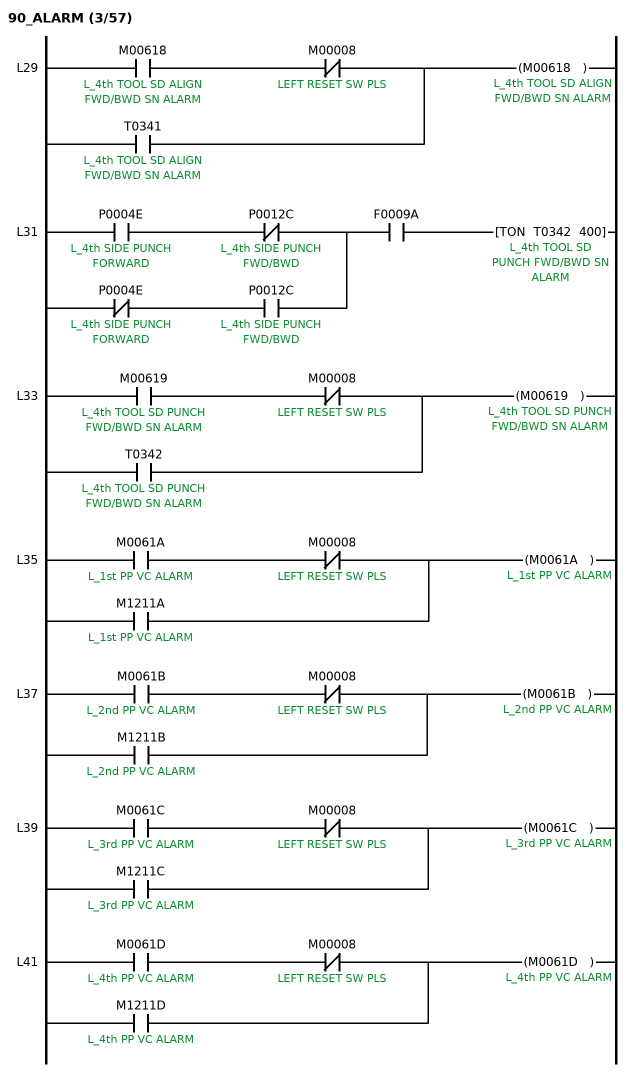
; L29
LOAD      M00618	// L_4th TOOL SD ALIGN FWD/BWD SN ALARM
AND NOT   M00008	// LEFT RESET SW PLS
OR        T0341	// L_4th TOOL SD ALIGN FWD/BWD SN ALARM
OUT       M00618	// L_4th TOOL SD ALIGN FWD/BWD SN ALARM
; L31
LOAD      P0004E	// L_4th SIDE PUNCH FORWARD
AND NOT   P0012C	// L_4th SIDE PUNCH FWD/BWD
LOAD NOT  P0004E	// L_4th SIDE PUNCH FORWARD
AND       P0012C	// L_4th SIDE PUNCH FWD/BWD
OR LOAD
AND       F0009A
TON       T0342 400	// L_4th TOOL SD PUNCH FWD/BWD SN ALARM
; L33
LOAD      M00619	// L_4th TOOL SD PUNCH FWD/BWD SN ALARM
AND NOT   M00008	// LEFT RESET SW PLS
OR        T0342	// L_4th TOOL SD PUNCH FWD/BWD SN ALARM
OUT       M00619	// L_4th TOOL SD PUNCH FWD/BWD SN ALARM
; L35
LOAD      M0061A	// L_1st PP VC ALARM
AND NOT   M00008	// LEFT RESET SW PLS
OR        M1211A	// L_1st PP VC ALARM
OUT       M0061A	// L_1st PP VC ALARM
; L37
LOAD      M0061B	// L_2nd PP VC ALARM
AND NOT   M00008	// LEFT RESET SW PLS
OR        M1211B	// L_2nd PP VC ALARM
OUT       M0061B	// L_2nd PP VC ALARM
; L39
LOAD      M0061C	// L_3rd PP VC ALARM
AND NOT   M00008	// LEFT RESET SW PLS
OR        M1211C	// L_3rd PP VC ALARM
OUT       M0061C	// L_3rd PP VC ALARM
; L41
LOAD      M0061D	// L_4th PP VC ALARM
AND NOT   M00008	// LEFT RESET SW PLS
OR        M1211D	// L_4th PP VC ALARM
OUT       M0061D	// L_4th PP VC ALARM

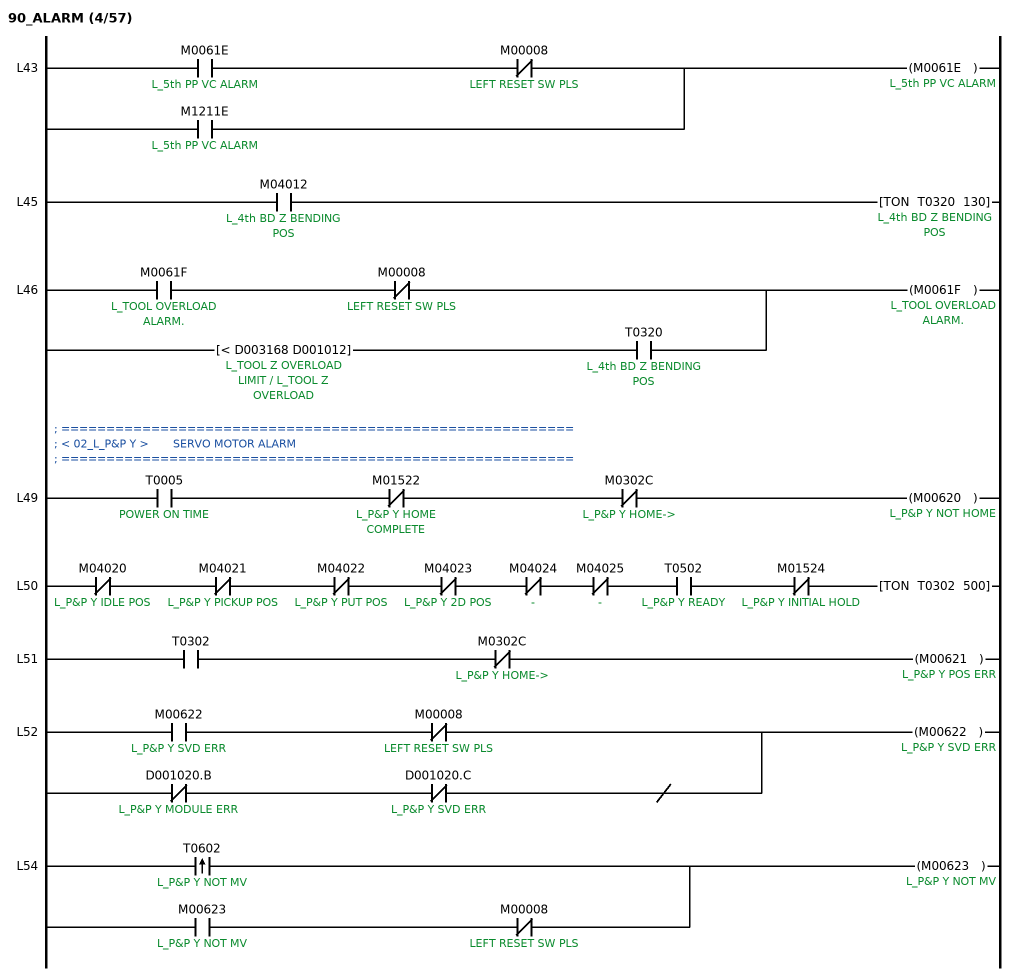
; L43
LOAD      M0061E	// L_5th PP VC ALARM
AND NOT   M00008	// LEFT RESET SW PLS
OR        M1211E	// L_5th PP VC ALARM
OUT       M0061E	// L_5th PP VC ALARM
; L45
LOAD      M04012	// L_4th BD Z BENDING POS
TON       T0320 130	// L_4th BD Z BENDING POS
; L46
LOAD      M0061F	// L_TOOL OVERLOAD ALARM.
AND NOT   M00008	// LEFT RESET SW PLS
LOAD<     D003168 D001012	// L_TOOL Z OVERLOAD LIMIT / L_TOOL Z OVERLOAD
AND       T0320	// L_4th BD Z BENDING POS
OR LOAD
OUT       M0061F	// L_TOOL OVERLOAD ALARM.
// =========================================================
// 
//        < 02_L_P&P Y >       SERVO MOTOR ALARM
// 
// =========================================================
; L49
LOAD      T0005	// POWER ON TIME
AND NOT   M01522	// L_P&P Y HOME COMPLETE
AND NOT   M0302C	// L_P&P Y HOME->
OUT       M00620	// L_P&P Y NOT HOME
; L50
LOAD NOT  M04020	// L_P&P Y IDLE POS
AND NOT   M04021	// L_P&P Y PICKUP POS
AND NOT   M04022	// L_P&P Y PUT POS
AND NOT   M04023	// L_P&P Y 2D POS
AND NOT   M04024	// -
AND NOT   M04025	// -
AND       T0502	// L_P&P Y READY
AND NOT   M01524	// L_P&P Y INITIAL HOLD
TON       T0302 500
; L51
LOAD      T0302
AND NOT   M0302C	// L_P&P Y HOME->
OUT       M00621	// L_P&P Y POS ERR
; L52
LOAD      M00622	// L_P&P Y SVD ERR
AND NOT   M00008	// LEFT RESET SW PLS
LOAD NOT  D001020.B	// L_P&P Y MODULE ERR
AND NOT   D001020.C	// L_P&P Y SVD ERR
NOT
OR LOAD
OUT       M00622	// L_P&P Y SVD ERR
; L54
LOADP     T0602	// L_P&P Y NOT MV
LOAD      M00623	// L_P&P Y NOT MV
AND NOT   M00008	// LEFT RESET SW PLS
OR LOAD
OUT       M00623	// L_P&P Y NOT MV

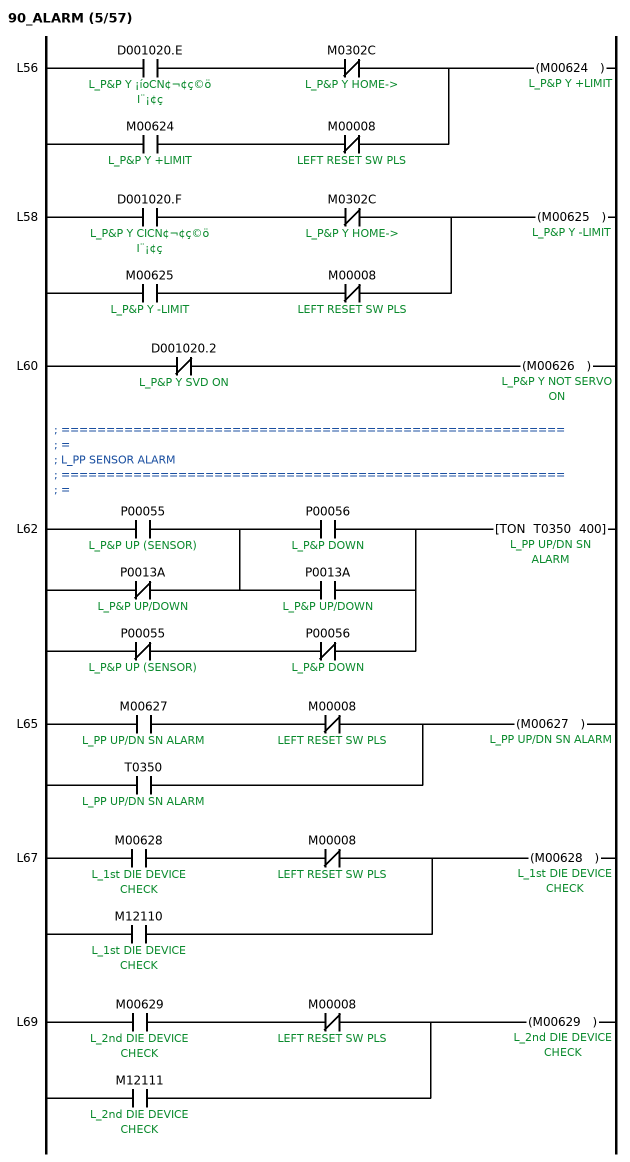
; L56
LOAD      D001020.E	// L_P&P Y ¡íoCN¢¬¢ç©öI¨¡¢ç
AND NOT   M0302C	// L_P&P Y HOME->
LOAD      M00624	// L_P&P Y +LIMIT
AND NOT   M00008	// LEFT RESET SW PLS
OR LOAD
OUT       M00624	// L_P&P Y +LIMIT
; L58
LOAD      D001020.F	// L_P&P Y CICN¢¬¢ç©öI¨¡¢ç
AND NOT   M0302C	// L_P&P Y HOME->
LOAD      M00625	// L_P&P Y -LIMIT
AND NOT   M00008	// LEFT RESET SW PLS
OR LOAD
OUT       M00625	// L_P&P Y -LIMIT
; L60
LOAD NOT  D001020.2	// L_P&P Y SVD ON
OUT       M00626	// L_P&P Y NOT SERVO ON
// =========================================================
// 
//       L_PP SENSOR ALARM
// 
// =========================================================
; L62
LOAD      P00055	// L_P&P UP (SENSOR)
OR NOT    P0013A	// L_P&P UP/DOWN
LOAD      P00056	// L_P&P DOWN
OR        P0013A	// L_P&P UP/DOWN
AND LOAD
LOAD NOT  P00055	// L_P&P UP (SENSOR)
AND NOT   P00056	// L_P&P DOWN
OR LOAD
TON       T0350 400	// L_PP UP/DN SN ALARM
; L65
LOAD      M00627	// L_PP UP/DN SN ALARM
AND NOT   M00008	// LEFT RESET SW PLS
OR        T0350	// L_PP UP/DN SN ALARM
OUT       M00627	// L_PP UP/DN SN ALARM
; L67
LOAD      M00628	// L_1st DIE DEVICE CHECK
AND NOT   M00008	// LEFT RESET SW PLS
OR        M12110	// L_1st DIE DEVICE CHECK
OUT       M00628	// L_1st DIE DEVICE CHECK
; L69
LOAD      M00629	// L_2nd DIE DEVICE CHECK
AND NOT   M00008	// LEFT RESET SW PLS
OR        M12111	// L_2nd DIE DEVICE CHECK
OUT       M00629	// L_2nd DIE DEVICE CHECK

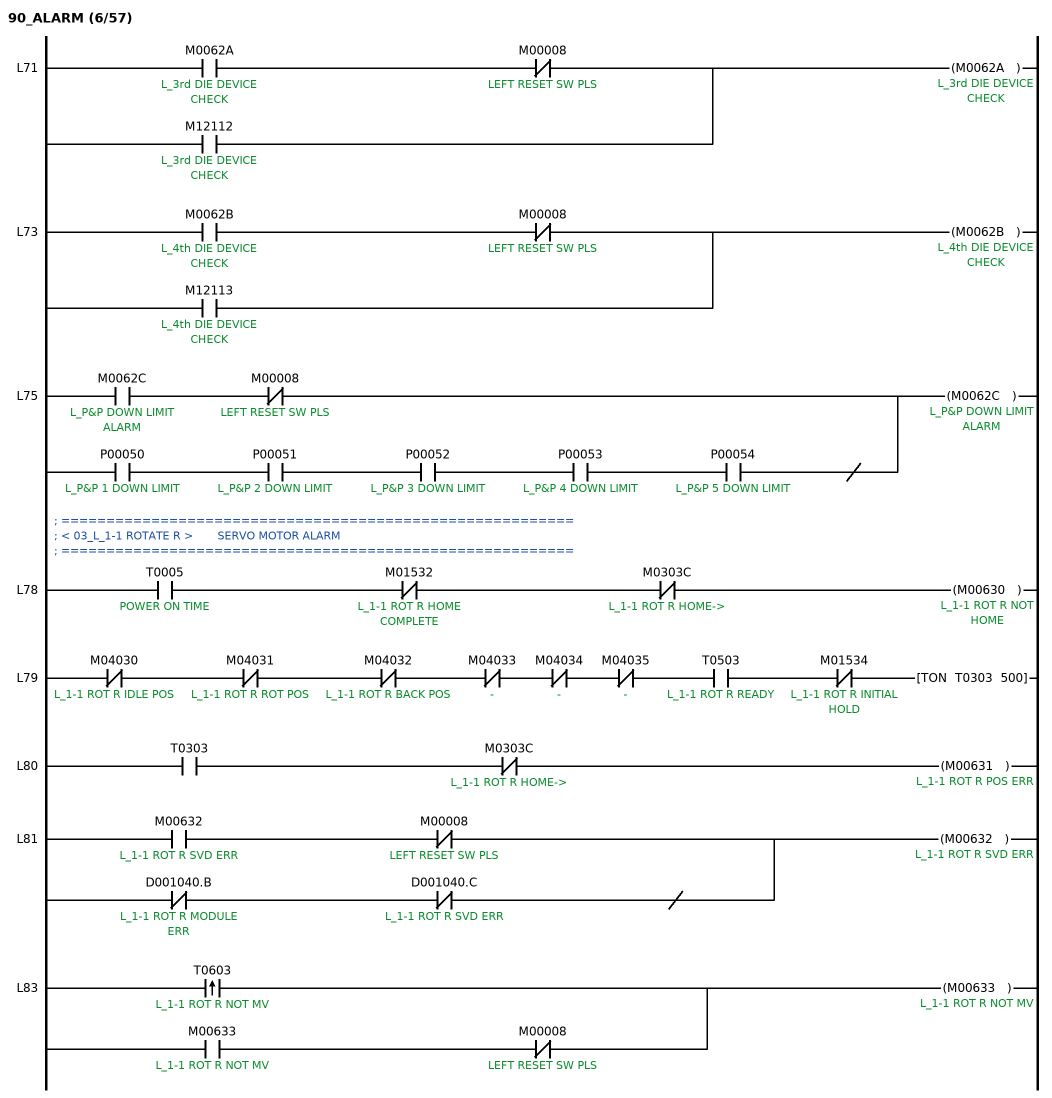
; L71
LOAD      M0062A	// L_3rd DIE DEVICE CHECK
AND NOT   M00008	// LEFT RESET SW PLS
OR        M12112	// L_3rd DIE DEVICE CHECK
OUT       M0062A	// L_3rd DIE DEVICE CHECK
; L73
LOAD      M0062B	// L_4th DIE DEVICE CHECK
AND NOT   M00008	// LEFT RESET SW PLS
OR        M12113	// L_4th DIE DEVICE CHECK
OUT       M0062B	// L_4th DIE DEVICE CHECK
; L75
LOAD      M0062C	// L_P&P DOWN LIMIT ALARM
AND NOT   M00008	// LEFT RESET SW PLS
LOAD      P00050	// L_P&P 1 DOWN LIMIT
AND       P00051	// L_P&P 2 DOWN LIMIT
AND       P00052	// L_P&P 3 DOWN LIMIT
AND       P00053	// L_P&P 4 DOWN LIMIT
AND       P00054	// L_P&P 5 DOWN LIMIT
NOT
OR LOAD
OUT       M0062C	// L_P&P DOWN LIMIT ALARM
// =========================================================
// 
//        < 03_L_1-1 ROTATE R >       SERVO MOTOR ALARM
// 
// =========================================================
; L78
LOAD      T0005	// POWER ON TIME
AND NOT   M01532	// L_1-1 ROT R HOME COMPLETE
AND NOT   M0303C	// L_1-1 ROT R HOME->
OUT       M00630	// L_1-1 ROT R NOT HOME
; L79
LOAD NOT  M04030	// L_1-1 ROT R IDLE POS
AND NOT   M04031	// L_1-1 ROT R ROT POS
AND NOT   M04032	// L_1-1 ROT R BACK POS
AND NOT   M04033	// -
AND NOT   M04034	// -
AND NOT   M04035	// -
AND       T0503	// L_1-1 ROT R READY
AND NOT   M01534	// L_1-1 ROT R INITIAL HOLD
TON       T0303 500
; L80
LOAD      T0303
AND NOT   M0303C	// L_1-1 ROT R HOME->
OUT       M00631	// L_1-1 ROT R POS ERR
; L81
LOAD      M00632	// L_1-1 ROT R SVD ERR
AND NOT   M00008	// LEFT RESET SW PLS
LOAD NOT  D001040.B	// L_1-1 ROT R MODULE ERR
AND NOT   D001040.C	// L_1-1 ROT R SVD ERR
NOT
OR LOAD
OUT       M00632	// L_1-1 ROT R SVD ERR
; L83
LOADP     T0603	// L_1-1 ROT R NOT MV
LOAD      M00633	// L_1-1 ROT R NOT MV
AND NOT   M00008	// LEFT RESET SW PLS
OR LOAD
OUT       M00633	// L_1-1 ROT R NOT MV

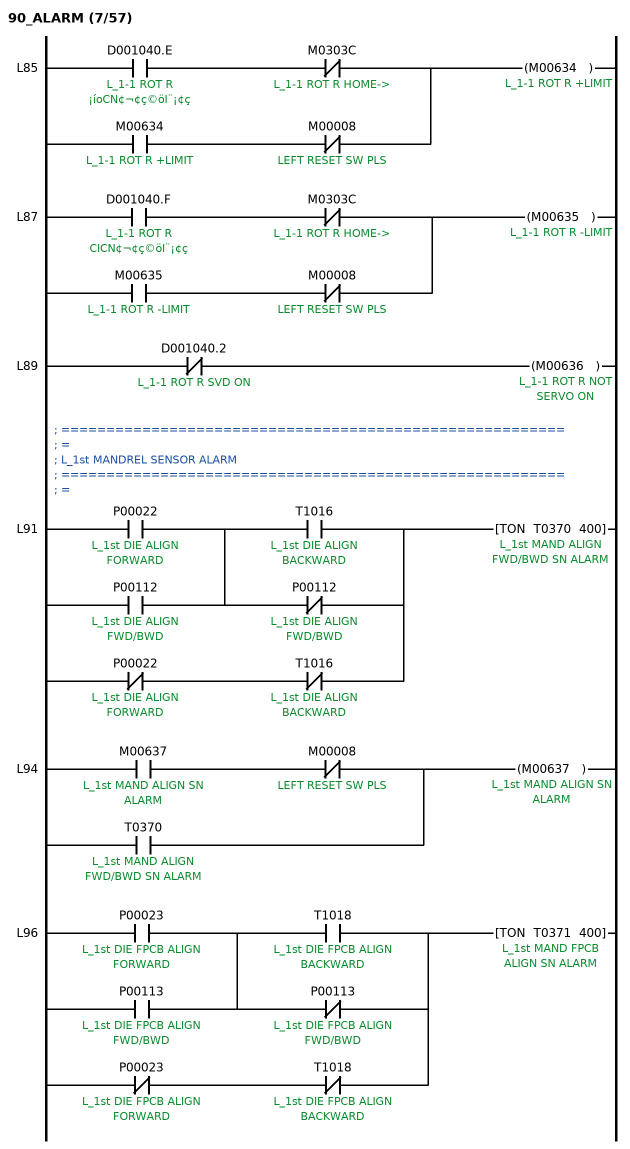
; L85
LOAD      D001040.E	// L_1-1 ROT R ¡íoCN¢¬¢ç©öI¨¡¢ç
AND NOT   M0303C	// L_1-1 ROT R HOME->
LOAD      M00634	// L_1-1 ROT R +LIMIT
AND NOT   M00008	// LEFT RESET SW PLS
OR LOAD
OUT       M00634	// L_1-1 ROT R +LIMIT
; L87
LOAD      D001040.F	// L_1-1 ROT R CICN¢¬¢ç©öI¨¡¢ç
AND NOT   M0303C	// L_1-1 ROT R HOME->
LOAD      M00635	// L_1-1 ROT R -LIMIT
AND NOT   M00008	// LEFT RESET SW PLS
OR LOAD
OUT       M00635	// L_1-1 ROT R -LIMIT
; L89
LOAD NOT  D001040.2	// L_1-1 ROT R SVD ON
OUT       M00636	// L_1-1 ROT R NOT SERVO ON
// =========================================================
// 
//        L_1st MANDREL SENSOR ALARM
// 
// =========================================================
; L91
LOAD      P00022	// L_1st DIE ALIGN FORWARD
OR        P00112	// L_1st DIE ALIGN FWD/BWD
LOAD      T1016	// L_1st DIE ALIGN BACKWARD
OR NOT    P00112	// L_1st DIE ALIGN FWD/BWD
AND LOAD
LOAD NOT  P00022	// L_1st DIE ALIGN FORWARD
AND NOT   T1016	// L_1st DIE ALIGN BACKWARD
OR LOAD
TON       T0370 400	// L_1st MAND ALIGN FWD/BWD SN ALARM
; L94
LOAD      M00637	// L_1st MAND ALIGN SN ALARM
AND NOT   M00008	// LEFT RESET SW PLS
OR        T0370	// L_1st MAND ALIGN FWD/BWD SN ALARM
OUT       M00637	// L_1st MAND ALIGN SN ALARM
; L96
LOAD      P00023	// L_1st DIE FPCB ALIGN FORWARD
OR        P00113	// L_1st DIE FPCB ALIGN FWD/BWD
LOAD      T1018	// L_1st DIE FPCB ALIGN BACKWARD
OR NOT    P00113	// L_1st DIE FPCB ALIGN FWD/BWD
AND LOAD
LOAD NOT  P00023	// L_1st DIE FPCB ALIGN FORWARD
AND NOT   T1018	// L_1st DIE FPCB ALIGN BACKWARD
OR LOAD
TON       T0371 400	// L_1st MAND FPCB ALIGN SN ALARM

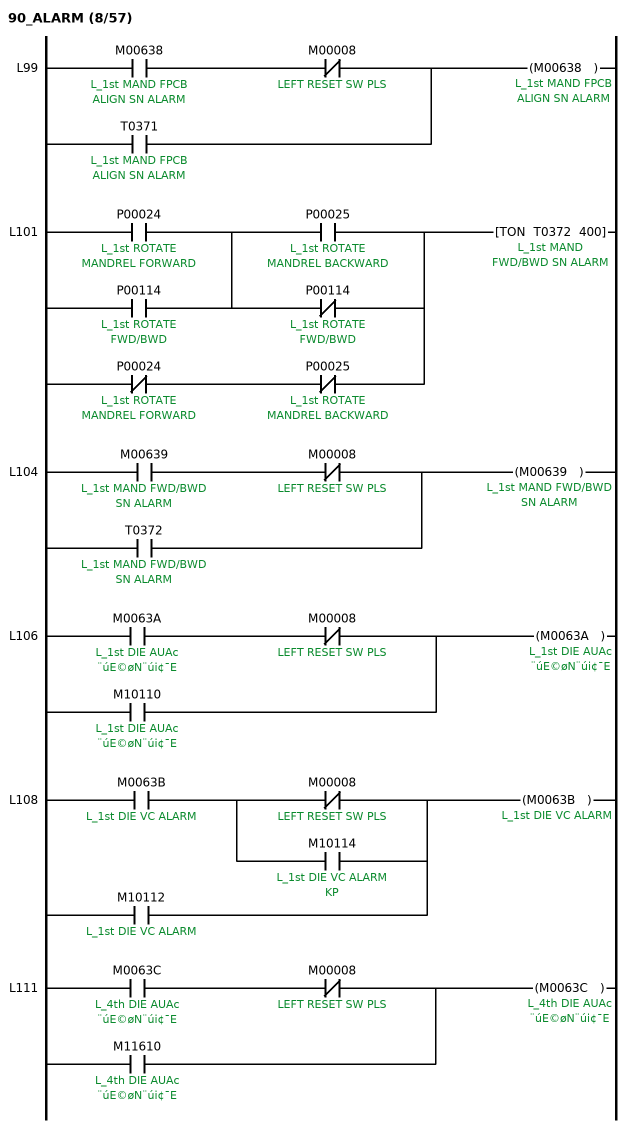
; L99
LOAD      M00638	// L_1st MAND FPCB ALIGN SN ALARM
AND NOT   M00008	// LEFT RESET SW PLS
OR        T0371	// L_1st MAND FPCB ALIGN SN ALARM
OUT       M00638	// L_1st MAND FPCB ALIGN SN ALARM
; L101
LOAD      P00024	// L_1st ROTATE MANDREL FORWARD
OR        P00114	// L_1st ROTATE FWD/BWD
LOAD      P00025	// L_1st ROTATE MANDREL BACKWARD
OR NOT    P00114	// L_1st ROTATE FWD/BWD
AND LOAD
LOAD NOT  P00024	// L_1st ROTATE MANDREL FORWARD
AND NOT   P00025	// L_1st ROTATE MANDREL BACKWARD
OR LOAD
TON       T0372 400	// L_1st MAND FWD/BWD SN ALARM
; L104
LOAD      M00639	// L_1st MAND FWD/BWD SN ALARM
AND NOT   M00008	// LEFT RESET SW PLS
OR        T0372	// L_1st MAND FWD/BWD SN ALARM
OUT       M00639	// L_1st MAND FWD/BWD SN ALARM
; L106
LOAD      M0063A	// L_1st DIE AUAc ¨úE©øN¨úi¢¯E
AND NOT   M00008	// LEFT RESET SW PLS
OR        M10110	// L_1st DIE AUAc ¨úE©øN¨úi¢¯E
OUT       M0063A	// L_1st DIE AUAc ¨úE©øN¨úi¢¯E
; L108
LOAD      M0063B	// L_1st DIE VC ALARM
LOAD NOT  M00008	// LEFT RESET SW PLS
OR        M10114	// L_1st DIE VC ALARM KP
AND LOAD
OR        M10112	// L_1st DIE VC ALARM
OUT       M0063B	// L_1st DIE VC ALARM
; L111
LOAD      M0063C	// L_4th DIE AUAc ¨úE©øN¨úi¢¯E
AND NOT   M00008	// LEFT RESET SW PLS
OR        M11610	// L_4th DIE AUAc ¨úE©øN¨úi¢¯E
OUT       M0063C	// L_4th DIE AUAc ¨úE©øN¨úi¢¯E

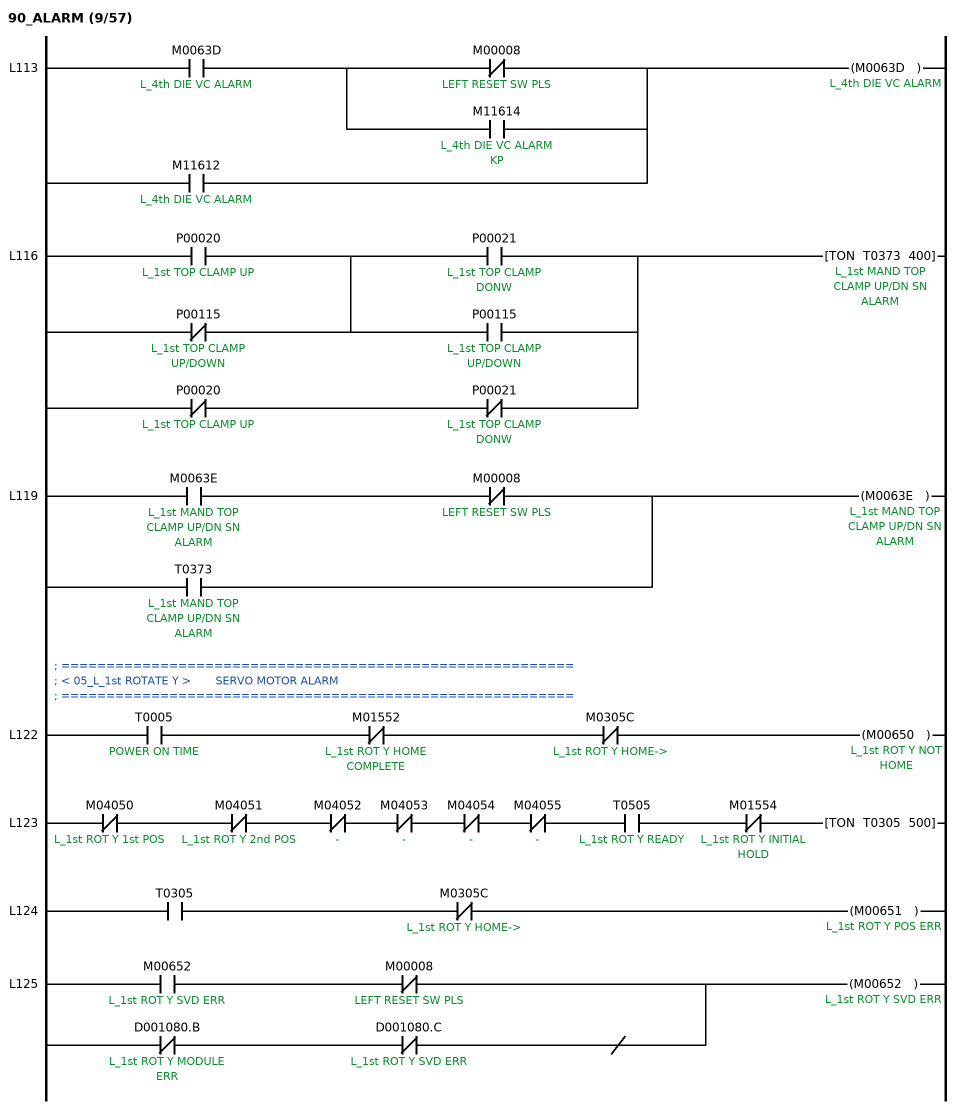
; L113
LOAD      M0063D	// L_4th DIE VC ALARM
LOAD NOT  M00008	// LEFT RESET SW PLS
OR        M11614	// L_4th DIE VC ALARM KP
AND LOAD
OR        M11612	// L_4th DIE VC ALARM
OUT       M0063D	// L_4th DIE VC ALARM
; L116
LOAD      P00020	// L_1st TOP CLAMP UP
OR NOT    P00115	// L_1st TOP CLAMP UP/DOWN
LOAD      P00021	// L_1st TOP CLAMP DONW
OR        P00115	// L_1st TOP CLAMP UP/DOWN
AND LOAD
LOAD NOT  P00020	// L_1st TOP CLAMP UP
AND NOT   P00021	// L_1st TOP CLAMP DONW
OR LOAD
TON       T0373 400	// L_1st MAND TOP CLAMP UP/DN SN ALARM
; L119
LOAD      M0063E	// L_1st MAND TOP CLAMP UP/DN SN ALARM
AND NOT   M00008	// LEFT RESET SW PLS
OR        T0373	// L_1st MAND TOP CLAMP UP/DN SN ALARM
OUT       M0063E	// L_1st MAND TOP CLAMP UP/DN SN ALARM
// =========================================================
// 
//        < 05_L_1st ROTATE Y >       SERVO MOTOR ALARM
// 
// =========================================================
; L122
LOAD      T0005	// POWER ON TIME
AND NOT   M01552	// L_1st ROT Y HOME COMPLETE
AND NOT   M0305C	// L_1st ROT Y HOME->
OUT       M00650	// L_1st ROT Y NOT HOME
; L123
LOAD NOT  M04050	// L_1st ROT Y 1st POS
AND NOT   M04051	// L_1st ROT Y 2nd POS
AND NOT   M04052	// -
AND NOT   M04053	// -
AND NOT   M04054	// -
AND NOT   M04055	// -
AND       T0505	// L_1st ROT Y READY
AND NOT   M01554	// L_1st ROT Y INITIAL HOLD
TON       T0305 500
; L124
LOAD      T0305
AND NOT   M0305C	// L_1st ROT Y HOME->
OUT       M00651	// L_1st ROT Y POS ERR
; L125
LOAD      M00652	// L_1st ROT Y SVD ERR
AND NOT   M00008	// LEFT RESET SW PLS
LOAD NOT  D001080.B	// L_1st ROT Y MODULE ERR
AND NOT   D001080.C	// L_1st ROT Y SVD ERR
NOT
OR LOAD
OUT       M00652	// L_1st ROT Y SVD ERR

